PROGRAM MAIN
VAR
END_VAR

AssignInsOuts();


A_System_Start();
IF gvl.bSystemStart THEN
	IF GVL.SystemRun THEN
		B_Machine_Center();
		C_Input_Conveyor();
		D_Stacker_Crane();
		E_Output_Conveyor();
	END_IF
    F_Faults();
END_IF

END_PROGRAM

(* stored: Version 1.1.0.1
   POU MAIN: Id {ae5f9f5b-fe60-4045-b87c-087f3fa0f3b8}, SpecialFunc None *)
